// TIA Portal V20 export
DATA_BLOCK "DriveDiagConfig"   // DB18
TITLE = DriveDiagConfig
AUTHOR : Siemens Digital Industries
FAMILY : LAF
NAME : LAF_DriveDiagConfigData
VERSION : 1.1
// Configuration data array for drive diagnostic
// stored: MemoryReserve 100
   VAR
      driveObjects : Array[0.."LAF_DRV_DIAG_NO_DO"] of "LAF_typeDriveDiagConfig";
   END_VAR
BEGIN
END_DATA_BLOCK
